TYPE ST_CyclicEventDetection :
STRUCT
  id: INT;
  submitted_in_last_invocation: BIT;
END_STRUCT
END_TYPE

(* stored: Version 1.1.0.1, ProductVersion 3.1.4024.9
   DUT ST_CyclicEventDetection: Id {572b5e63-3823-479f-8ebe-a6103ff37c23} *)
